FUNCTION_BLOCK CAerationActuators (* Composite Function Block Type *)
  (* Standard: 61499-2 *)
  (* Version 0.0, 11/16/2023, SESA371406, Schneider Electric, template *)
  PACKAGE SE.Nereda;
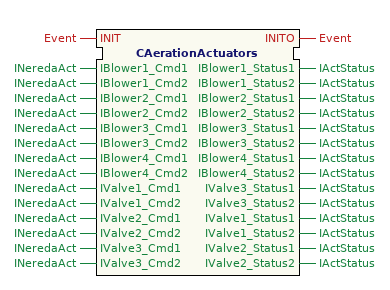
  EVENT_INPUT
    INIT;
  END_EVENT
  EVENT_OUTPUT
    INITO;
  END_EVENT
  SOCKETS
    IBlower1_Cmd1 : INeredaAct;
    IBlower1_Cmd2 : INeredaAct;
    IBlower2_Cmd1 : INeredaAct;
    IBlower2_Cmd2 : INeredaAct;
    IBlower3_Cmd1 : INeredaAct;
    IBlower3_Cmd2 : INeredaAct;
    IBlower4_Cmd1 : INeredaAct;
    IBlower4_Cmd2 : INeredaAct;
    IValve1_Cmd1 : INeredaAct;
    IValve1_Cmd2 : INeredaAct;
    IValve2_Cmd1 : INeredaAct;
    IValve2_Cmd2 : INeredaAct;
    IValve3_Cmd1 : INeredaAct;
    IValve3_Cmd2 : INeredaAct;
  END_SOCKETS
  PLUGS
    IBlower1_Status1 : IActStatus;
    IBlower1_Status2 : IActStatus;
    IBlower2_Status1 : IActStatus;
    IBlower2_Status2 : IActStatus;
    IBlower3_Status1 : IActStatus;
    IBlower3_Status2 : IActStatus;
    IBlower4_Status1 : IActStatus;
    IBlower4_Status2 : IActStatus;
    IValve3_Status1 : IActStatus;
    IValve3_Status2 : IActStatus;
    IValve1_Status1 : IActStatus;
    IValve1_Status2 : IActStatus;
    IValve2_Status1 : IActStatus;
    IValve2_Status2 : IActStatus;
  END_PLUGS
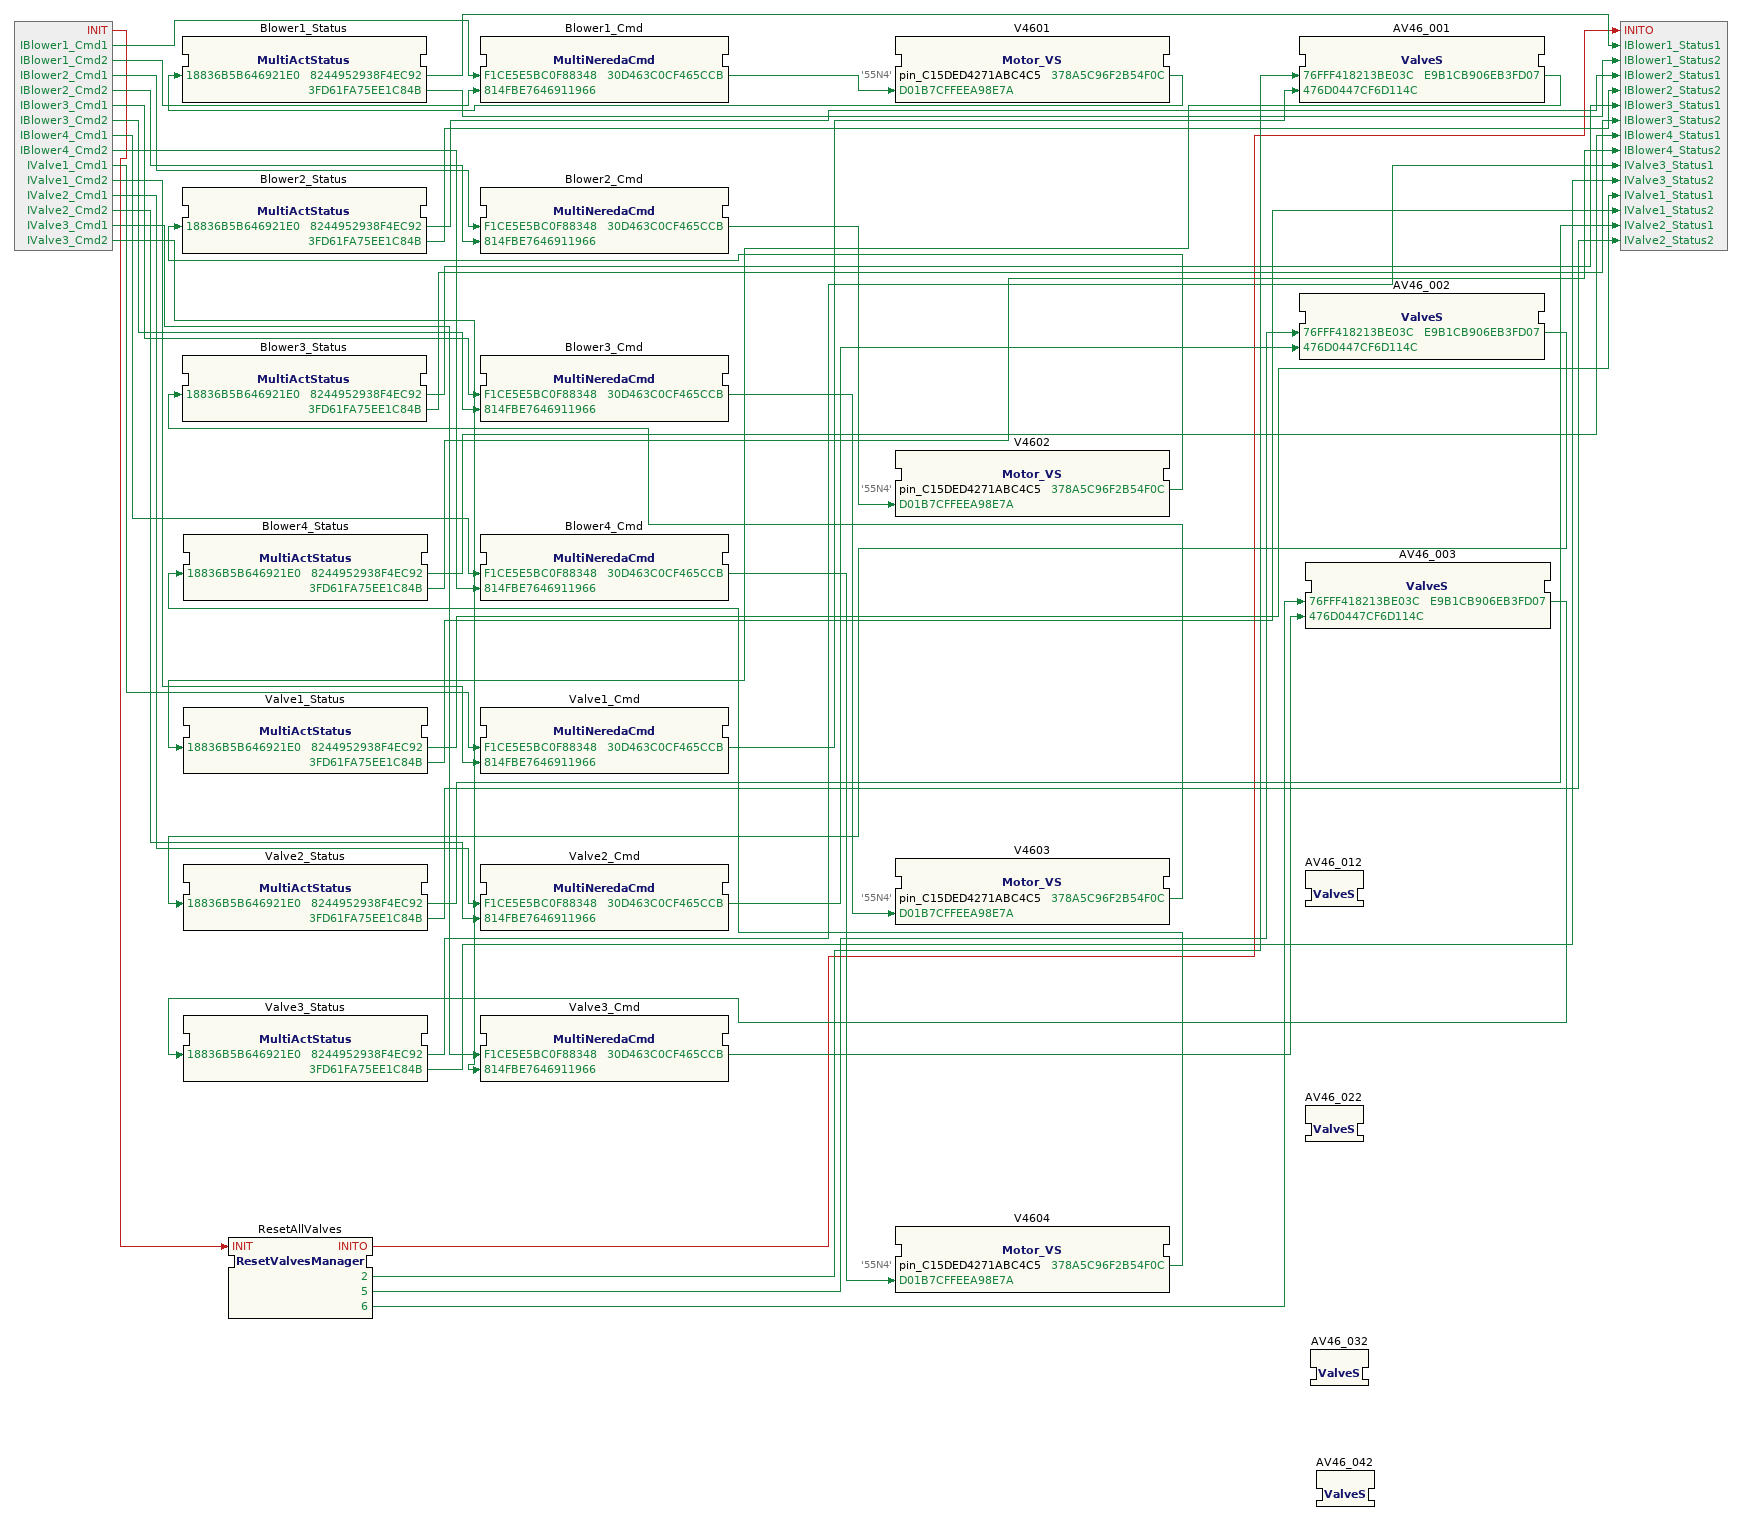
  (* 01 - FUNCTIONNAL INPUT INTERFACE *)
  (* 00 - INITIALIZATION *)
  (* 05 - LOGIC *)
  (* 06 - HMI INTERFACE *)
  (* 03 - FIELD INTERFACE *)
  (* 02 - FUNCTIONNAL OUTPUT INTERFACE *)
  (* Actuators Status *)
  (* 04 - CHILDREN *)
  (* 4A - TYPICALS *)
  (* Actuators Command *)
  (* Reset All Actuators *)
  FBS
    ResetAllValves : ResetValvesManager;
    Blower1_Status : MultiActStatus;
    Blower2_Status : MultiActStatus;
    Blower3_Status : MultiActStatus;
    Blower1_Cmd : MultiNeredaCmd;
    Blower2_Cmd : MultiNeredaCmd;
    Blower3_Cmd : MultiNeredaCmd;
    V4601 : Motor_VS(pin_C15DED4271ABC4C5 := '55N4');
    V4602 : Motor_VS(pin_C15DED4271ABC4C5 := '55N4');
    V4603 : Motor_VS(pin_C15DED4271ABC4C5 := '55N4');
    V4604 : Motor_VS(pin_C15DED4271ABC4C5 := '55N4');
    Blower4_Status : MultiActStatus;
    Blower4_Cmd : MultiNeredaCmd;
    AV46_001 : ValveS;
    AV46_002 : ValveS;
    AV46_003 : ValveS;
    Valve1_Status : MultiActStatus;
    Valve2_Status : MultiActStatus;
    Valve1_Cmd : MultiNeredaCmd;
    Valve2_Cmd : MultiNeredaCmd;
    Valve3_Status : MultiActStatus;
    Valve3_Cmd : MultiNeredaCmd;
    AV46_012 : ValveS;
    AV46_022 : ValveS;
    AV46_032 : ValveS;
    AV46_042 : ValveS;
  END_FBS
  EVENT_CONNECTIONS
    INIT TO ResetAllValves.INIT;
    ResetAllValves.INITO TO INITO;
  END_CONNECTIONS
  ADAPTER_CONNECTIONS
    IBlower1_Cmd1 TO Blower1_Cmd.F1CE5E5BC0F88348;
    IBlower1_Cmd2 TO Blower1_Cmd.814FBE7646911966;
    IBlower2_Cmd1 TO Blower2_Cmd.F1CE5E5BC0F88348;
    IBlower2_Cmd2 TO Blower2_Cmd.814FBE7646911966;
    IBlower3_Cmd1 TO Blower3_Cmd.F1CE5E5BC0F88348;
    IBlower3_Cmd2 TO Blower3_Cmd.814FBE7646911966;
    Blower1_Status.8244952938F4EC92 TO IBlower1_Status1;
    Blower1_Status.3FD61FA75EE1C84B TO IBlower1_Status2;
    Blower2_Status.8244952938F4EC92 TO IBlower2_Status1;
    Blower2_Status.3FD61FA75EE1C84B TO IBlower2_Status2;
    Blower3_Status.8244952938F4EC92 TO IBlower3_Status1;
    Blower3_Status.3FD61FA75EE1C84B TO IBlower3_Status2;
    Blower1_Cmd.30D463C0CF465CCB TO V4601.D01B7CFFEEA98E7A;
    Blower2_Cmd.30D463C0CF465CCB TO V4602.D01B7CFFEEA98E7A;
    Blower3_Cmd.30D463C0CF465CCB TO V4603.D01B7CFFEEA98E7A;
    Blower4_Cmd.30D463C0CF465CCB TO V4604.D01B7CFFEEA98E7A;
    IBlower4_Cmd1 TO Blower4_Cmd.F1CE5E5BC0F88348;
    IBlower4_Cmd2 TO Blower4_Cmd.814FBE7646911966;
    Blower4_Status.8244952938F4EC92 TO IBlower4_Status1;
    Blower4_Status.3FD61FA75EE1C84B TO IBlower4_Status2;
    V4601.378A5C96F2B54F0C TO Blower1_Status.18836B5B646921E0;
    V4602.378A5C96F2B54F0C TO Blower2_Status.18836B5B646921E0;
    V4603.378A5C96F2B54F0C TO Blower3_Status.18836B5B646921E0;
    V4604.378A5C96F2B54F0C TO Blower4_Status.18836B5B646921E0;
    ResetAllValves.2 TO AV46_001.76FFF418213BE03C;
    ResetAllValves.5 TO AV46_002.76FFF418213BE03C;
    ResetAllValves.6 TO AV46_003.76FFF418213BE03C;
    Valve1_Cmd.30D463C0CF465CCB TO AV46_001.476D0447CF6D114C;
    Valve2_Cmd.30D463C0CF465CCB TO AV46_002.476D0447CF6D114C;
    Valve3_Cmd.30D463C0CF465CCB TO AV46_003.476D0447CF6D114C;
    AV46_001.E9B1CB906EB3FD07 TO Valve1_Status.18836B5B646921E0;
    AV46_002.E9B1CB906EB3FD07 TO Valve2_Status.18836B5B646921E0;
    AV46_003.E9B1CB906EB3FD07 TO Valve3_Status.18836B5B646921E0;
    IValve1_Cmd1 TO Valve1_Cmd.F1CE5E5BC0F88348;
    IValve1_Cmd2 TO Valve1_Cmd.814FBE7646911966;
    IValve2_Cmd1 TO Valve2_Cmd.F1CE5E5BC0F88348;
    IValve2_Cmd2 TO Valve2_Cmd.814FBE7646911966;
    IValve3_Cmd1 TO Valve3_Cmd.F1CE5E5BC0F88348;
    IValve3_Cmd2 TO Valve3_Cmd.814FBE7646911966;
    Valve1_Status.8244952938F4EC92 TO IValve1_Status1;
    Valve1_Status.3FD61FA75EE1C84B TO IValve1_Status2;
    Valve2_Status.8244952938F4EC92 TO IValve2_Status1;
    Valve2_Status.3FD61FA75EE1C84B TO IValve2_Status2;
    Valve3_Status.8244952938F4EC92 TO IValve3_Status1;
    Valve3_Status.3FD61FA75EE1C84B TO IValve3_Status2;
  END_CONNECTIONS
END_FUNCTION_BLOCK
